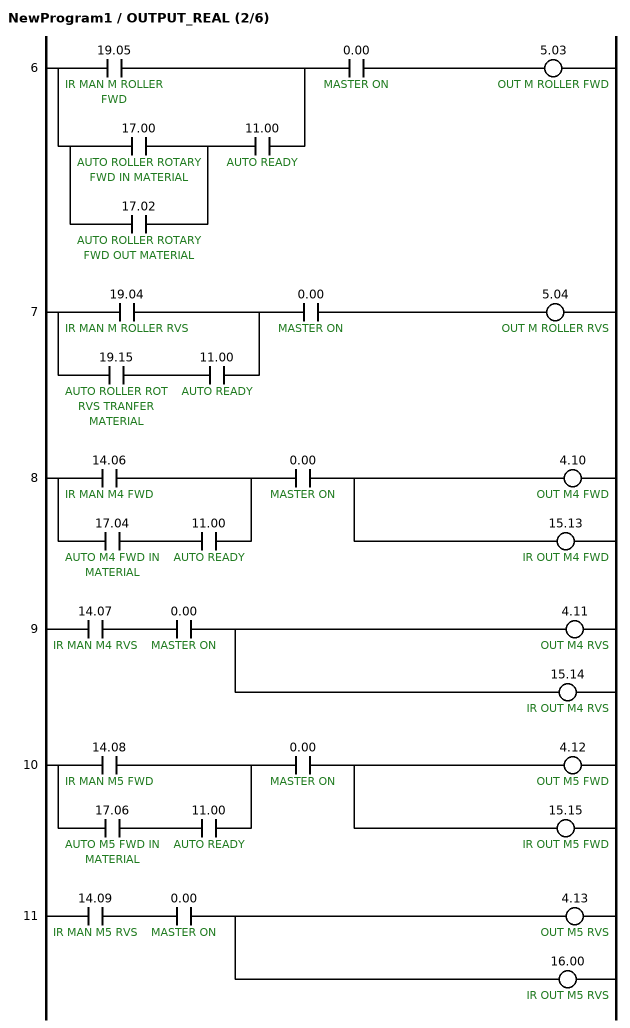
; [picture p24: NewProgram1 / OUTPUT_REAL, rungs 6-11]
; rung 6
LD 19.05  ; IR MAN M ROLLER FWD
LD 17.00  ; AUTO ROLLER ROTARY FWD IN MATERIAL
OR 17.02  ; AUTO ROLLER ROTARY FWD OUT MATERIAL
AND 11.00  ; AUTO READY
ORLD
AND 0.00  ; MASTER ON
OUT 5.03  ; OUT M ROLLER FWD
; rung 7
LD 19.04  ; IR MAN M ROLLER RVS
LD 19.15  ; AUTO ROLLER ROT RVS TRANFER MATERIAL
AND 11.00  ; AUTO READY
ORLD
AND 0.00  ; MASTER ON
OUT 5.04  ; OUT M ROLLER RVS
; rung 8
LD 14.06  ; IR MAN M4 FWD
LD 17.04  ; AUTO M4 FWD IN MATERIAL
AND 11.00  ; AUTO READY
ORLD
AND 0.00  ; MASTER ON
OUT 4.10  ; OUT M4 FWD
OUT 15.13  ; IR OUT M4 FWD
; rung 9
LD 14.07  ; IR MAN M4 RVS
AND 0.00  ; MASTER ON
OUT 4.11  ; OUT M4 RVS
OUT 15.14  ; IR OUT M4 RVS
; rung 10
LD 14.08  ; IR MAN M5 FWD
LD 17.06  ; AUTO M5 FWD IN MATERIAL
AND 11.00  ; AUTO READY
ORLD
AND 0.00  ; MASTER ON
OUT 4.12  ; OUT M5 FWD
OUT 15.15  ; IR OUT M5 FWD
; rung 11
LD 14.09  ; IR MAN M5 RVS
AND 0.00  ; MASTER ON
OUT 4.13  ; OUT M5 RVS
OUT 16.00  ; IR OUT M5 RVS

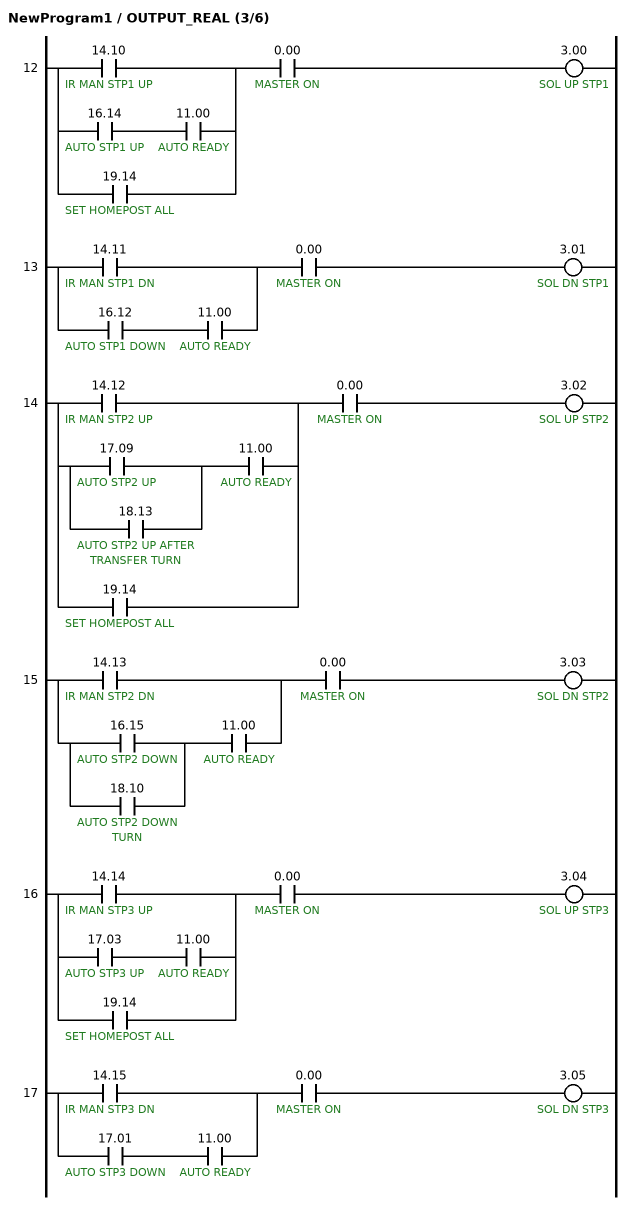
; rung 12
LD 14.10  ; IR MAN STP1 UP
LD 16.14  ; AUTO STP1 UP
AND 11.00  ; AUTO READY
ORLD
OR 19.14  ; SET HOMEPOST ALL
AND 0.00  ; MASTER ON
OUT 3.00  ; SOL UP STP1
; rung 13
LD 14.11  ; IR MAN STP1 DN
LD 16.12  ; AUTO STP1 DOWN
AND 11.00  ; AUTO READY
ORLD
AND 0.00  ; MASTER ON
OUT 3.01  ; SOL DN STP1
; rung 14
LD 14.12  ; IR MAN STP2 UP
LD 17.09  ; AUTO STP2 UP
OR 18.13  ; AUTO STP2 UP AFTER TRANSFER TURN
AND 11.00  ; AUTO READY
ORLD
OR 19.14  ; SET HOMEPOST ALL
AND 0.00  ; MASTER ON
OUT 3.02  ; SOL UP STP2
; rung 15
LD 14.13  ; IR MAN STP2 DN
LD 16.15  ; AUTO STP2 DOWN
OR 18.10  ; AUTO STP2 DOWN TURN
AND 11.00  ; AUTO READY
ORLD
AND 0.00  ; MASTER ON
OUT 3.03  ; SOL DN STP2
; rung 16
LD 14.14  ; IR MAN STP3 UP
LD 17.03  ; AUTO STP3 UP
AND 11.00  ; AUTO READY
ORLD
OR 19.14  ; SET HOMEPOST ALL
AND 0.00  ; MASTER ON
OUT 3.04  ; SOL UP STP3
; rung 17
LD 14.15  ; IR MAN STP3 DN
LD 17.01  ; AUTO STP3 DOWN
AND 11.00  ; AUTO READY
ORLD
AND 0.00  ; MASTER ON
OUT 3.05  ; SOL DN STP3

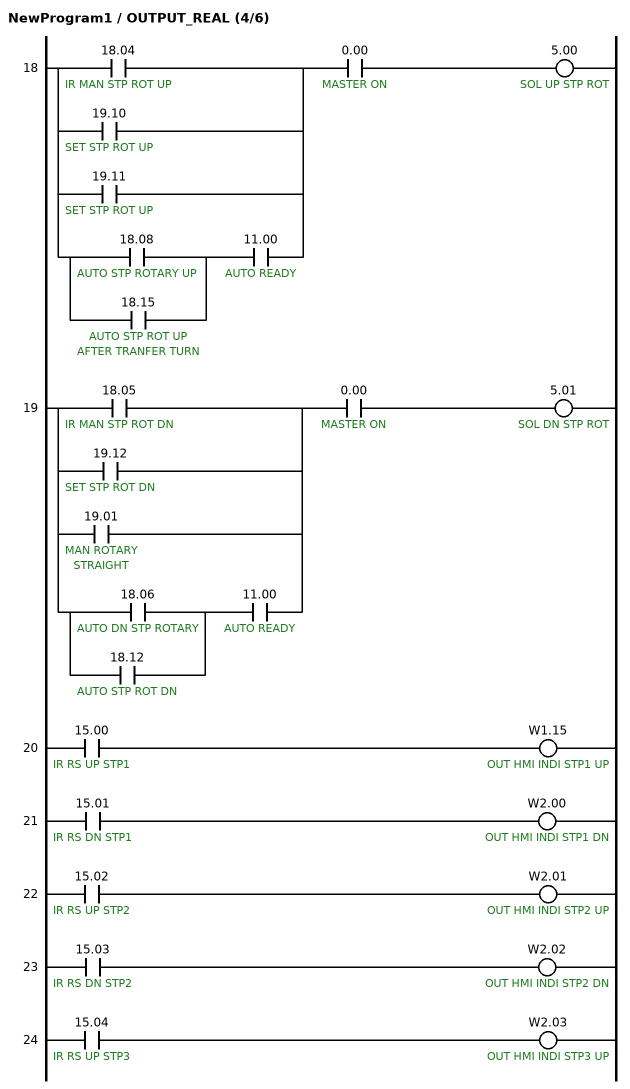
; rung 18
LD 18.04  ; IR MAN STP ROT UP
OR 19.10  ; SET STP ROT UP
OR 19.11  ; SET STP ROT UP
LD 18.08  ; AUTO STP ROTARY UP
OR 18.15  ; AUTO STP ROT UP AFTER TRANFER TURN
AND 11.00  ; AUTO READY
ORLD
AND 0.00  ; MASTER ON
OUT 5.00  ; SOL UP STP ROT
; rung 19
LD 18.05  ; IR MAN STP ROT DN
OR 19.12  ; SET STP ROT DN
OR 19.01  ; MAN ROTARY STRAIGHT
LD 18.06  ; AUTO DN STP ROTARY
OR 18.12  ; AUTO STP ROT DN
AND 11.00  ; AUTO READY
ORLD
AND 0.00  ; MASTER ON
OUT 5.01  ; SOL DN STP ROT
; rung 20
LD 15.00  ; IR RS UP STP1
OUT W1.15  ; OUT HMI INDI STP1 UP
; rung 21
LD 15.01  ; IR RS DN STP1
OUT W2.00  ; OUT HMI INDI STP1 DN
; rung 22
LD 15.02  ; IR RS UP STP2
OUT W2.01  ; OUT HMI INDI STP2 UP
; rung 23
LD 15.03  ; IR RS DN STP2
OUT W2.02  ; OUT HMI INDI STP2 DN
; rung 24
LD 15.04  ; IR RS UP STP3
OUT W2.03  ; OUT HMI INDI STP3 UP

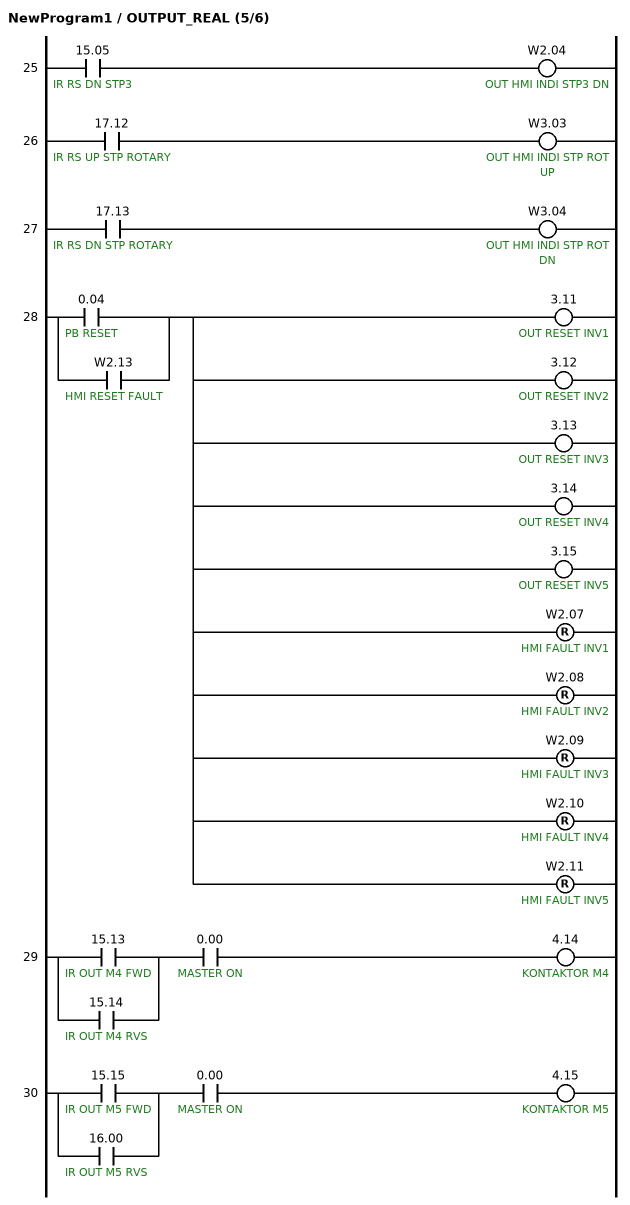
; rung 25
LD 15.05  ; IR RS DN STP3
OUT W2.04  ; OUT HMI INDI STP3 DN
; rung 26
LD 17.12  ; IR RS UP STP ROTARY
OUT W3.03  ; OUT HMI INDI STP ROT UP
; rung 27
LD 17.13  ; IR RS DN STP ROTARY
OUT W3.04  ; OUT HMI INDI STP ROT DN
; rung 28
LD 0.04  ; PB RESET
OR W2.13  ; HMI RESET FAULT
OUT 3.11  ; OUT RESET INV1
OUT 3.12  ; OUT RESET INV2
OUT 3.13  ; OUT RESET INV3
OUT 3.14  ; OUT RESET INV4
OUT 3.15  ; OUT RESET INV5
RSET W2.07  ; HMI FAULT INV1
RSET W2.08  ; HMI FAULT INV2
RSET W2.09  ; HMI FAULT INV3
RSET W2.10  ; HMI FAULT INV4
RSET W2.11  ; HMI FAULT INV5
; rung 29
LD 15.13  ; IR OUT M4 FWD
OR 15.14  ; IR OUT M4 RVS
AND 0.00  ; MASTER ON
OUT 4.14  ; KONTAKTOR M4
; rung 30
LD 15.15  ; IR OUT M5 FWD
OR 16.00  ; IR OUT M5 RVS
AND 0.00  ; MASTER ON
OUT 4.15  ; KONTAKTOR M5

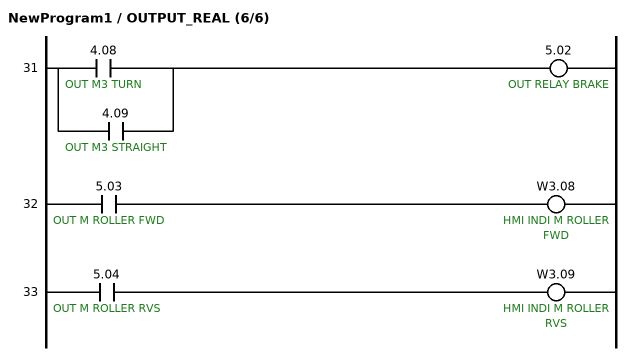
; rung 31
LD 4.08  ; OUT M3 TURN
OR 4.09  ; OUT M3 STRAIGHT
OUT 5.02  ; OUT RELAY BRAKE
; rung 32
LD 5.03  ; OUT M ROLLER FWD
OUT W3.08  ; HMI INDI M ROLLER FWD
; rung 33
LD 5.04  ; OUT M ROLLER RVS
OUT W3.09  ; HMI INDI M ROLLER RVS

### Section INPUT_REAL

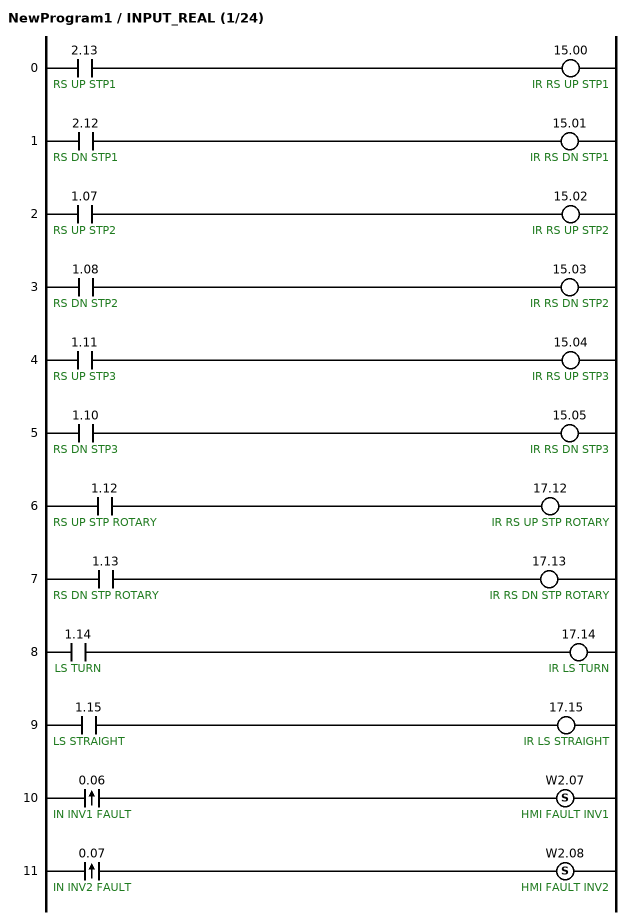
; rung 0
LD 2.13  ; RS UP STP1
OUT 15.00  ; IR RS UP STP1
; rung 1
LD 2.12  ; RS DN STP1
OUT 15.01  ; IR RS DN STP1
; rung 2
LD 1.07  ; RS UP STP2
OUT 15.02  ; IR RS UP STP2
; rung 3
LD 1.08  ; RS DN STP2
OUT 15.03  ; IR RS DN STP2
; rung 4
LD 1.11  ; RS UP STP3
OUT 15.04  ; IR RS UP STP3
; rung 5
LD 1.10  ; RS DN STP3
OUT 15.05  ; IR RS DN STP3
; rung 6
LD 1.12  ; RS UP STP ROTARY
OUT 17.12  ; IR RS UP STP ROTARY
; rung 7
LD 1.13  ; RS DN STP ROTARY
OUT 17.13  ; IR RS DN STP ROTARY
; rung 8
LD 1.14  ; LS TURN
OUT 17.14  ; IR LS TURN
; rung 9
LD 1.15  ; LS STRAIGHT
OUT 17.15  ; IR LS STRAIGHT
; rung 10
@LD 0.06  ; IN INV1 FAULT
SET W2.07  ; HMI FAULT INV1
; rung 11
@LD 0.07  ; IN INV2 FAULT
SET W2.08  ; HMI FAULT INV2

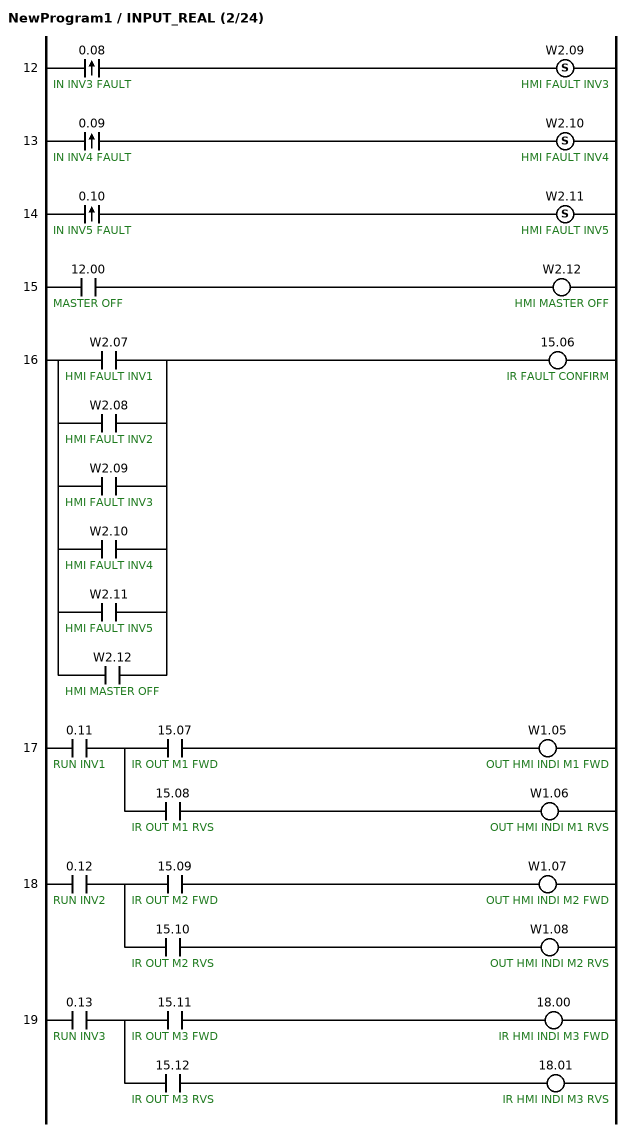
; rung 12
@LD 0.08  ; IN INV3 FAULT
SET W2.09  ; HMI FAULT INV3
; rung 13
@LD 0.09  ; IN INV4 FAULT
SET W2.10  ; HMI FAULT INV4
; rung 14
@LD 0.10  ; IN INV5 FAULT
SET W2.11  ; HMI FAULT INV5
; rung 15
LD 12.00  ; MASTER OFF
OUT W2.12  ; HMI MASTER OFF
; rung 16
LD W2.07  ; HMI FAULT INV1
OR W2.08  ; HMI FAULT INV2
OR W2.09  ; HMI FAULT INV3
OR W2.10  ; HMI FAULT INV4
OR W2.11  ; HMI FAULT INV5
OR W2.12  ; HMI MASTER OFF
OUT 15.06  ; IR FAULT CONFIRM
; rung 17
LD 0.11  ; RUN INV1
OUT TR0
AND 15.07  ; IR OUT M1 FWD
OUT W1.05  ; OUT HMI INDI M1 FWD
LD TR0
AND 15.08  ; IR OUT M1 RVS
OUT W1.06  ; OUT HMI INDI M1 RVS
; rung 18
LD 0.12  ; RUN INV2
OUT TR0
AND 15.09  ; IR OUT M2 FWD
OUT W1.07  ; OUT HMI INDI M2 FWD
LD TR0
AND 15.10  ; IR OUT M2 RVS
OUT W1.08  ; OUT HMI INDI M2 RVS
; rung 19
LD 0.13  ; RUN INV3
OUT TR0
AND 15.11  ; IR OUT M3 FWD
OUT 18.00  ; IR HMI INDI M3 FWD
LD TR0
AND 15.12  ; IR OUT M3 RVS
OUT 18.01  ; IR HMI INDI M3 RVS

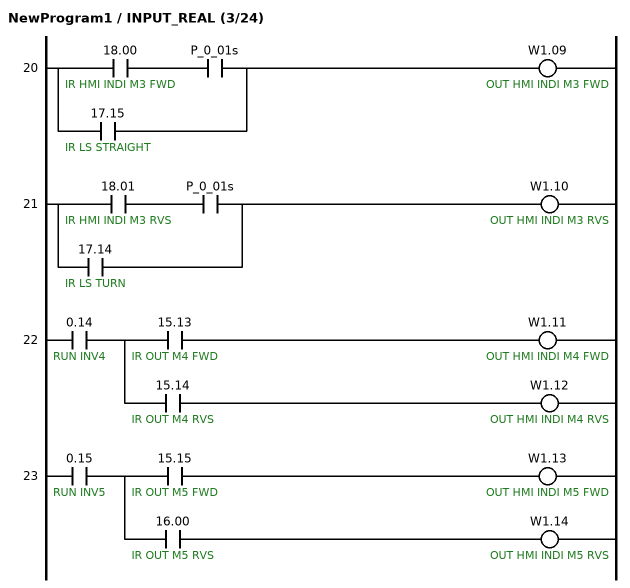
; rung 20
LD 18.00  ; IR HMI INDI M3 FWD
AND P_0_01s
OR 17.15  ; IR LS STRAIGHT
OUT W1.09  ; OUT HMI INDI M3 FWD
; rung 21
LD 18.01  ; IR HMI INDI M3 RVS
AND P_0_01s
OR 17.14  ; IR LS TURN
OUT W1.10  ; OUT HMI INDI M3 RVS
; rung 22
LD 0.14  ; RUN INV4
OUT TR0
AND 15.13  ; IR OUT M4 FWD
OUT W1.11  ; OUT HMI INDI M4 FWD
LD TR0
AND 15.14  ; IR OUT M4 RVS
OUT W1.12  ; OUT HMI INDI M4 RVS
; rung 23
LD 0.15  ; RUN INV5
OUT TR0
AND 15.15  ; IR OUT M5 FWD
OUT W1.13  ; OUT HMI INDI M5 FWD
LD TR0
AND 16.00  ; IR OUT M5 RVS
OUT W1.14  ; OUT HMI INDI M5 RVS

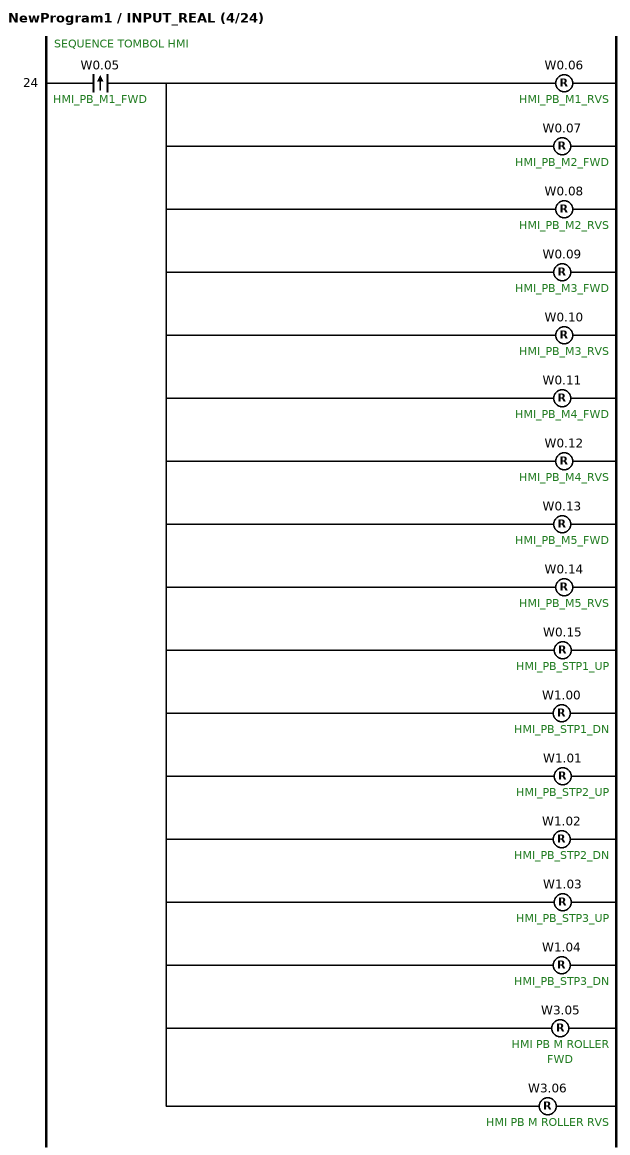
; rung 24: SEQUENCE TOMBOL HMI
@LD W0.05  ; HMI_PB_M1_FWD
RSET W0.06  ; HMI_PB_M1_RVS
RSET W0.07  ; HMI_PB_M2_FWD
RSET W0.08  ; HMI_PB_M2_RVS
RSET W0.09  ; HMI_PB_M3_FWD
RSET W0.10  ; HMI_PB_M3_RVS
RSET W0.11  ; HMI_PB_M4_FWD
RSET W0.12  ; HMI_PB_M4_RVS
RSET W0.13  ; HMI_PB_M5_FWD
RSET W0.14  ; HMI_PB_M5_RVS
RSET W0.15  ; HMI_PB_STP1_UP
RSET W1.00  ; HMI_PB_STP1_DN
RSET W1.01  ; HMI_PB_STP2_UP
RSET W1.02  ; HMI_PB_STP2_DN
RSET W1.03  ; HMI_PB_STP3_UP
RSET W1.04  ; HMI_PB_STP3_DN
RSET W3.05  ; HMI PB M ROLLER FWD
RSET W3.06  ; HMI PB M ROLLER RVS

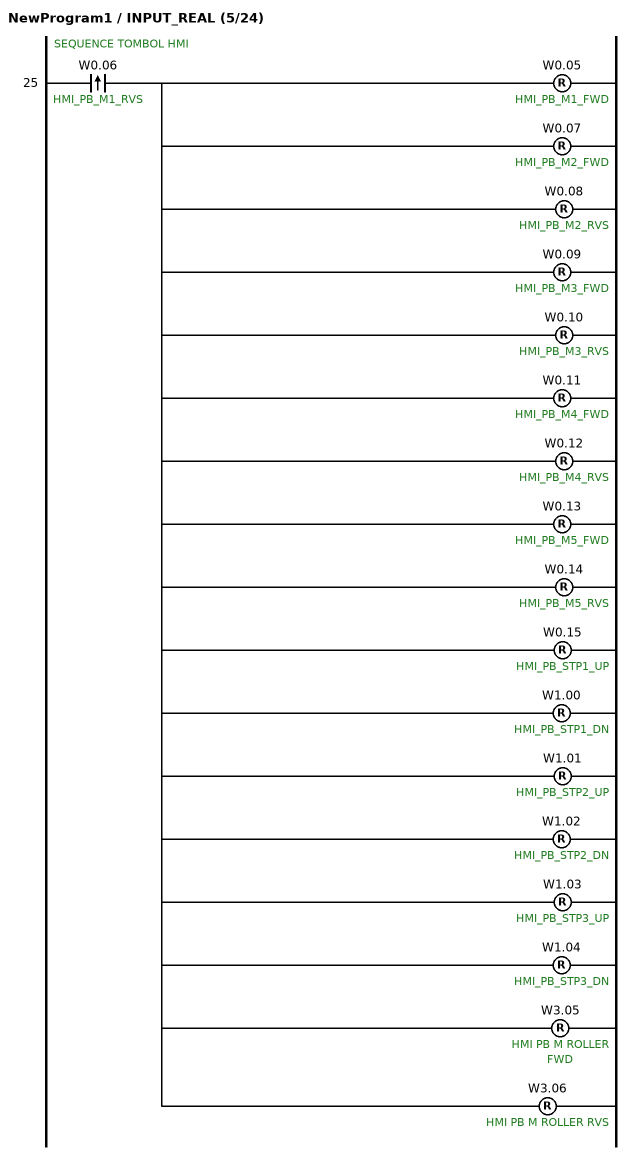
; rung 25: SEQUENCE TOMBOL HMI
@LD W0.06  ; HMI_PB_M1_RVS
RSET W0.05  ; HMI_PB_M1_FWD
RSET W0.07  ; HMI_PB_M2_FWD
RSET W0.08  ; HMI_PB_M2_RVS
RSET W0.09  ; HMI_PB_M3_FWD
RSET W0.10  ; HMI_PB_M3_RVS
RSET W0.11  ; HMI_PB_M4_FWD
RSET W0.12  ; HMI_PB_M4_RVS
RSET W0.13  ; HMI_PB_M5_FWD
RSET W0.14  ; HMI_PB_M5_RVS
RSET W0.15  ; HMI_PB_STP1_UP
RSET W1.00  ; HMI_PB_STP1_DN
RSET W1.01  ; HMI_PB_STP2_UP
RSET W1.02  ; HMI_PB_STP2_DN
RSET W1.03  ; HMI_PB_STP3_UP
RSET W1.04  ; HMI_PB_STP3_DN
RSET W3.05  ; HMI PB M ROLLER FWD
RSET W3.06  ; HMI PB M ROLLER RVS

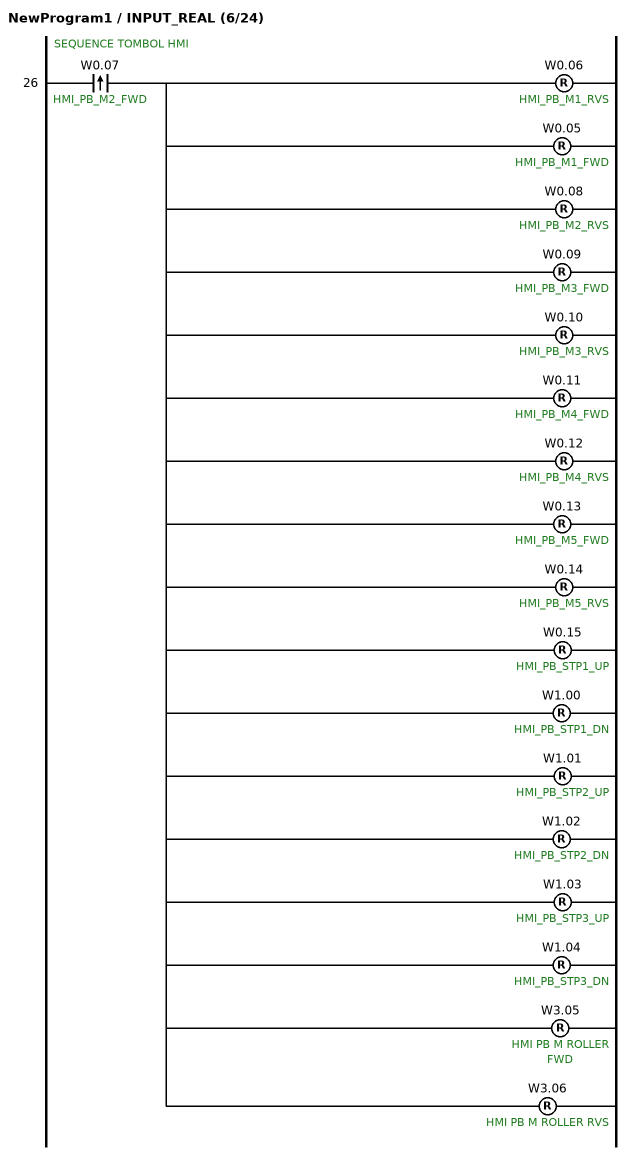
; rung 26: SEQUENCE TOMBOL HMI
@LD W0.07  ; HMI_PB_M2_FWD
RSET W0.06  ; HMI_PB_M1_RVS
RSET W0.05  ; HMI_PB_M1_FWD
RSET W0.08  ; HMI_PB_M2_RVS
RSET W0.09  ; HMI_PB_M3_FWD
RSET W0.10  ; HMI_PB_M3_RVS
RSET W0.11  ; HMI_PB_M4_FWD
RSET W0.12  ; HMI_PB_M4_RVS
RSET W0.13  ; HMI_PB_M5_FWD
RSET W0.14  ; HMI_PB_M5_RVS
RSET W0.15  ; HMI_PB_STP1_UP
RSET W1.00  ; HMI_PB_STP1_DN
RSET W1.01  ; HMI_PB_STP2_UP
RSET W1.02  ; HMI_PB_STP2_DN
RSET W1.03  ; HMI_PB_STP3_UP
RSET W1.04  ; HMI_PB_STP3_DN
RSET W3.05  ; HMI PB M ROLLER FWD
RSET W3.06  ; HMI PB M ROLLER RVS

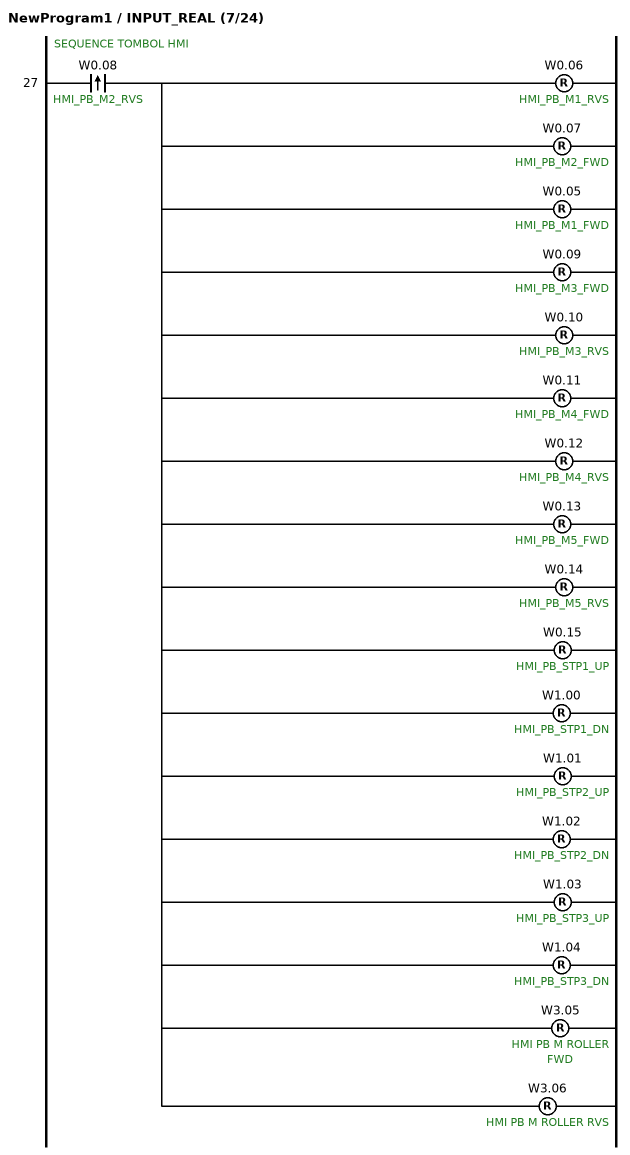
; rung 27: SEQUENCE TOMBOL HMI
@LD W0.08  ; HMI_PB_M2_RVS
RSET W0.06  ; HMI_PB_M1_RVS
RSET W0.07  ; HMI_PB_M2_FWD
RSET W0.05  ; HMI_PB_M1_FWD
RSET W0.09  ; HMI_PB_M3_FWD
RSET W0.10  ; HMI_PB_M3_RVS
RSET W0.11  ; HMI_PB_M4_FWD
RSET W0.12  ; HMI_PB_M4_RVS
RSET W0.13  ; HMI_PB_M5_FWD
RSET W0.14  ; HMI_PB_M5_RVS
RSET W0.15  ; HMI_PB_STP1_UP
RSET W1.00  ; HMI_PB_STP1_DN
RSET W1.01  ; HMI_PB_STP2_UP
RSET W1.02  ; HMI_PB_STP2_DN
RSET W1.03  ; HMI_PB_STP3_UP
RSET W1.04  ; HMI_PB_STP3_DN
RSET W3.05  ; HMI PB M ROLLER FWD
RSET W3.06  ; HMI PB M ROLLER RVS

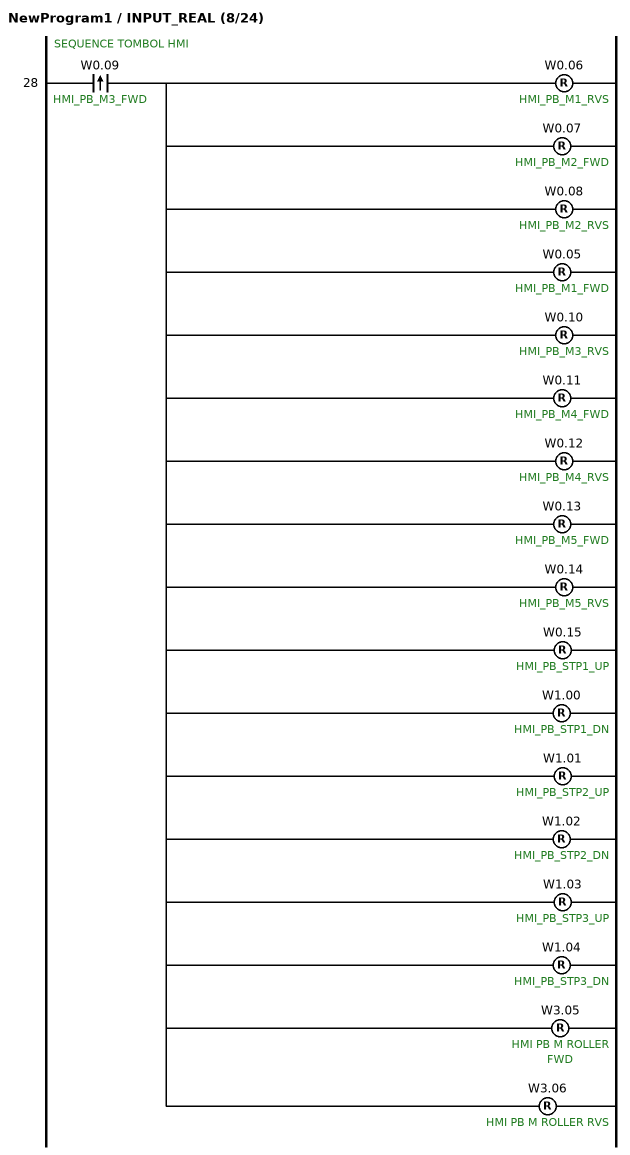
; rung 28: SEQUENCE TOMBOL HMI
@LD W0.09  ; HMI_PB_M3_FWD
RSET W0.06  ; HMI_PB_M1_RVS
RSET W0.07  ; HMI_PB_M2_FWD
RSET W0.08  ; HMI_PB_M2_RVS
RSET W0.05  ; HMI_PB_M1_FWD
RSET W0.10  ; HMI_PB_M3_RVS
RSET W0.11  ; HMI_PB_M4_FWD
RSET W0.12  ; HMI_PB_M4_RVS
RSET W0.13  ; HMI_PB_M5_FWD
RSET W0.14  ; HMI_PB_M5_RVS
RSET W0.15  ; HMI_PB_STP1_UP
RSET W1.00  ; HMI_PB_STP1_DN
RSET W1.01  ; HMI_PB_STP2_UP
RSET W1.02  ; HMI_PB_STP2_DN
RSET W1.03  ; HMI_PB_STP3_UP
RSET W1.04  ; HMI_PB_STP3_DN
RSET W3.05  ; HMI PB M ROLLER FWD
RSET W3.06  ; HMI PB M ROLLER RVS

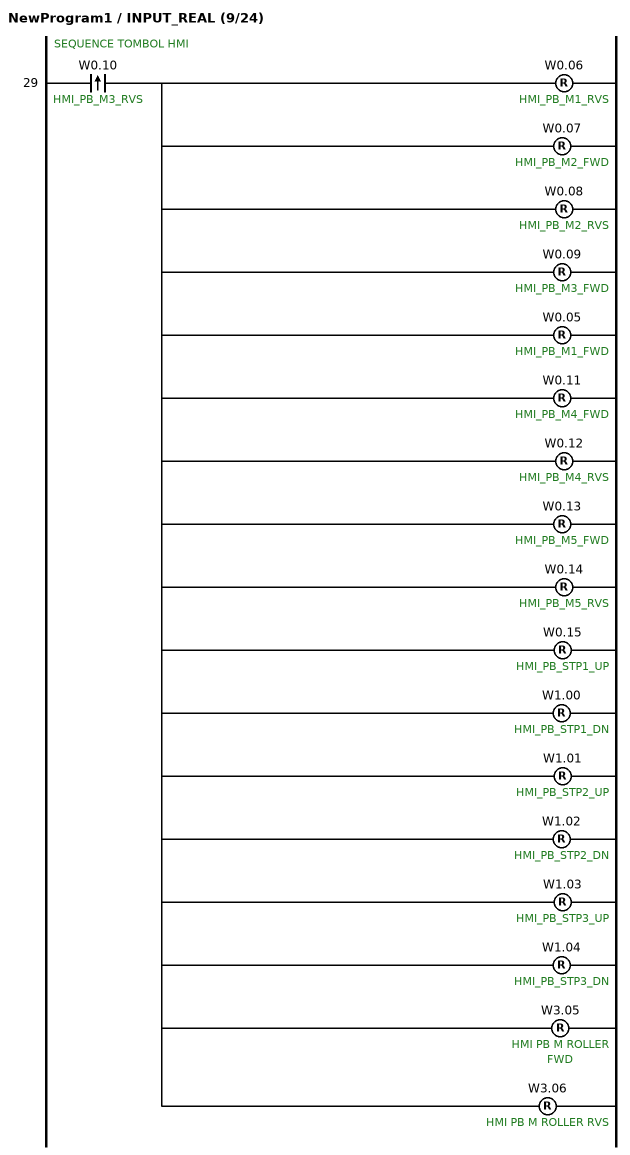
; rung 29: SEQUENCE TOMBOL HMI
@LD W0.10  ; HMI_PB_M3_RVS
RSET W0.06  ; HMI_PB_M1_RVS
RSET W0.07  ; HMI_PB_M2_FWD
RSET W0.08  ; HMI_PB_M2_RVS
RSET W0.09  ; HMI_PB_M3_FWD
RSET W0.05  ; HMI_PB_M1_FWD
RSET W0.11  ; HMI_PB_M4_FWD
RSET W0.12  ; HMI_PB_M4_RVS
RSET W0.13  ; HMI_PB_M5_FWD
RSET W0.14  ; HMI_PB_M5_RVS
RSET W0.15  ; HMI_PB_STP1_UP
RSET W1.00  ; HMI_PB_STP1_DN
RSET W1.01  ; HMI_PB_STP2_UP
RSET W1.02  ; HMI_PB_STP2_DN
RSET W1.03  ; HMI_PB_STP3_UP
RSET W1.04  ; HMI_PB_STP3_DN
RSET W3.05  ; HMI PB M ROLLER FWD
RSET W3.06  ; HMI PB M ROLLER RVS

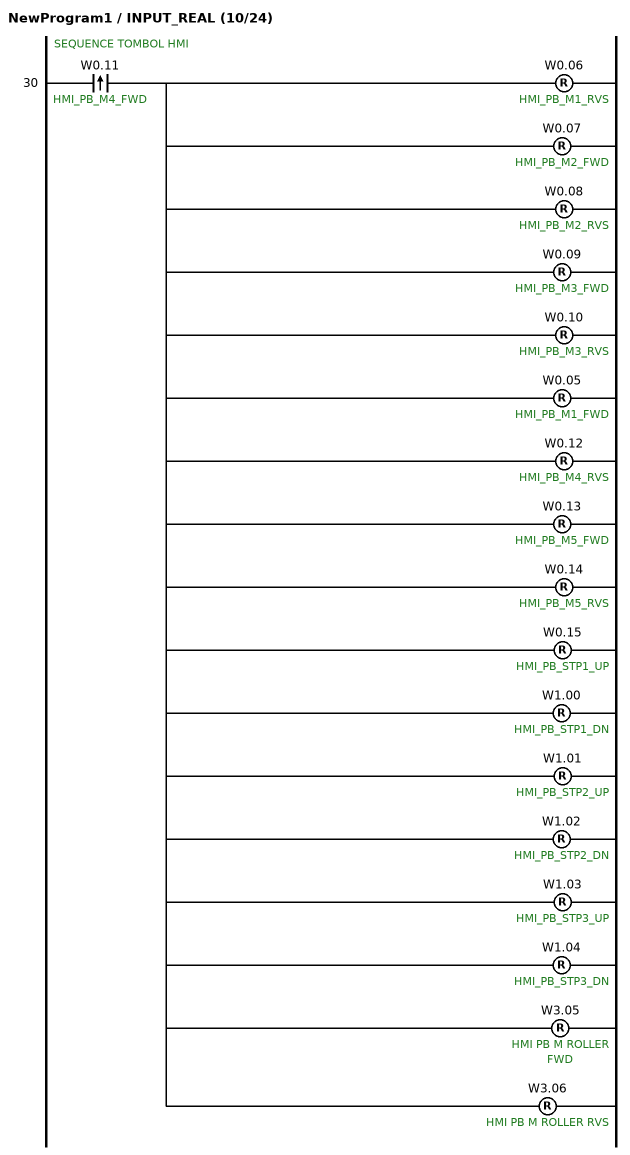
; rung 30: SEQUENCE TOMBOL HMI
@LD W0.11  ; HMI_PB_M4_FWD
RSET W0.06  ; HMI_PB_M1_RVS
RSET W0.07  ; HMI_PB_M2_FWD
RSET W0.08  ; HMI_PB_M2_RVS
RSET W0.09  ; HMI_PB_M3_FWD
RSET W0.10  ; HMI_PB_M3_RVS
RSET W0.05  ; HMI_PB_M1_FWD
RSET W0.12  ; HMI_PB_M4_RVS
RSET W0.13  ; HMI_PB_M5_FWD
RSET W0.14  ; HMI_PB_M5_RVS
RSET W0.15  ; HMI_PB_STP1_UP
RSET W1.00  ; HMI_PB_STP1_DN
RSET W1.01  ; HMI_PB_STP2_UP
RSET W1.02  ; HMI_PB_STP2_DN
RSET W1.03  ; HMI_PB_STP3_UP
RSET W1.04  ; HMI_PB_STP3_DN
RSET W3.05  ; HMI PB M ROLLER FWD
RSET W3.06  ; HMI PB M ROLLER RVS

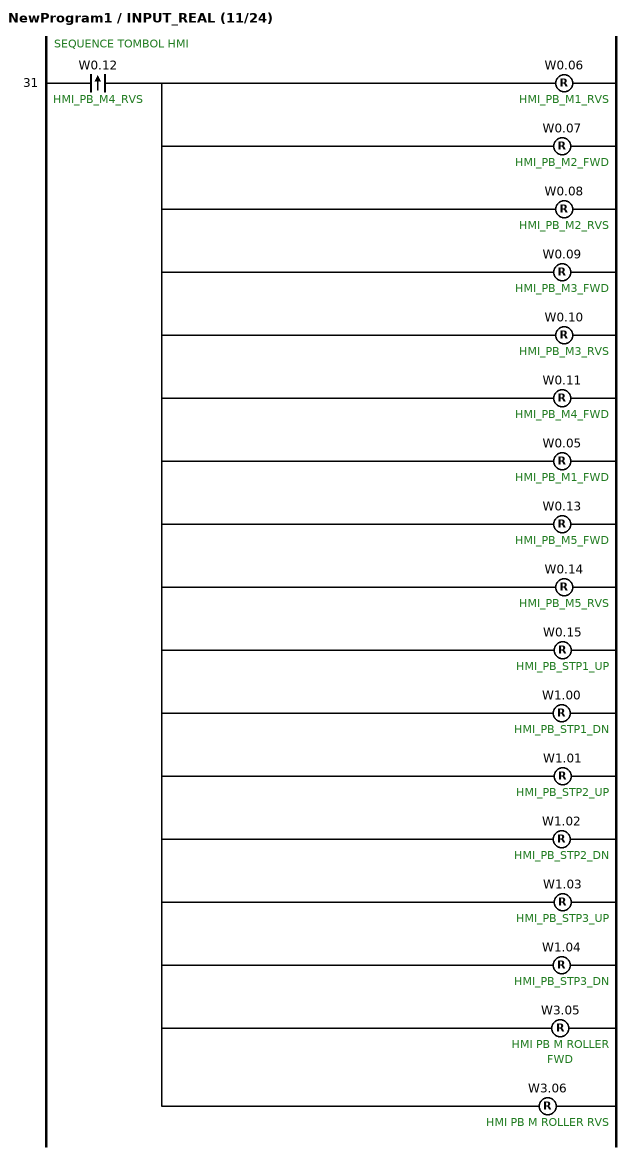
; rung 31: SEQUENCE TOMBOL HMI
@LD W0.12  ; HMI_PB_M4_RVS
RSET W0.06  ; HMI_PB_M1_RVS
RSET W0.07  ; HMI_PB_M2_FWD
RSET W0.08  ; HMI_PB_M2_RVS
RSET W0.09  ; HMI_PB_M3_FWD
RSET W0.10  ; HMI_PB_M3_RVS
RSET W0.11  ; HMI_PB_M4_FWD
RSET W0.05  ; HMI_PB_M1_FWD
RSET W0.13  ; HMI_PB_M5_FWD
RSET W0.14  ; HMI_PB_M5_RVS
RSET W0.15  ; HMI_PB_STP1_UP
RSET W1.00  ; HMI_PB_STP1_DN
RSET W1.01  ; HMI_PB_STP2_UP
RSET W1.02  ; HMI_PB_STP2_DN
RSET W1.03  ; HMI_PB_STP3_UP
RSET W1.04  ; HMI_PB_STP3_DN
RSET W3.05  ; HMI PB M ROLLER FWD
RSET W3.06  ; HMI PB M ROLLER RVS

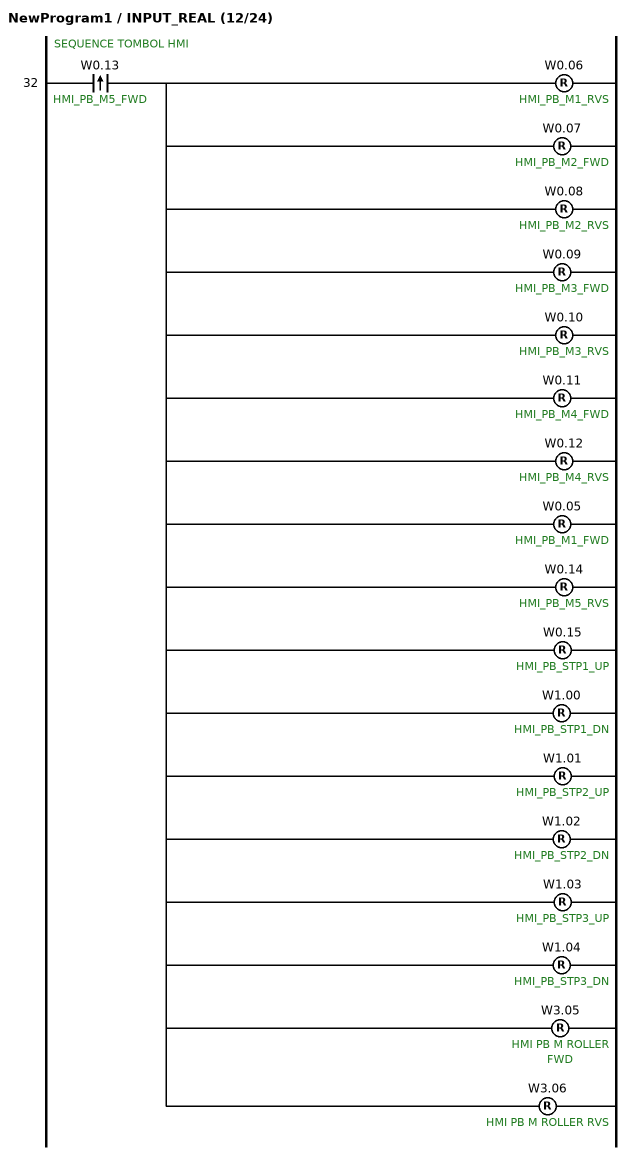
; rung 32: SEQUENCE TOMBOL HMI
@LD W0.13  ; HMI_PB_M5_FWD
RSET W0.06  ; HMI_PB_M1_RVS
RSET W0.07  ; HMI_PB_M2_FWD
RSET W0.08  ; HMI_PB_M2_RVS
RSET W0.09  ; HMI_PB_M3_FWD
RSET W0.10  ; HMI_PB_M3_RVS
RSET W0.11  ; HMI_PB_M4_FWD
RSET W0.12  ; HMI_PB_M4_RVS
RSET W0.05  ; HMI_PB_M1_FWD
RSET W0.14  ; HMI_PB_M5_RVS
RSET W0.15  ; HMI_PB_STP1_UP
RSET W1.00  ; HMI_PB_STP1_DN
RSET W1.01  ; HMI_PB_STP2_UP
RSET W1.02  ; HMI_PB_STP2_DN
RSET W1.03  ; HMI_PB_STP3_UP
RSET W1.04  ; HMI_PB_STP3_DN
RSET W3.05  ; HMI PB M ROLLER FWD
RSET W3.06  ; HMI PB M ROLLER RVS

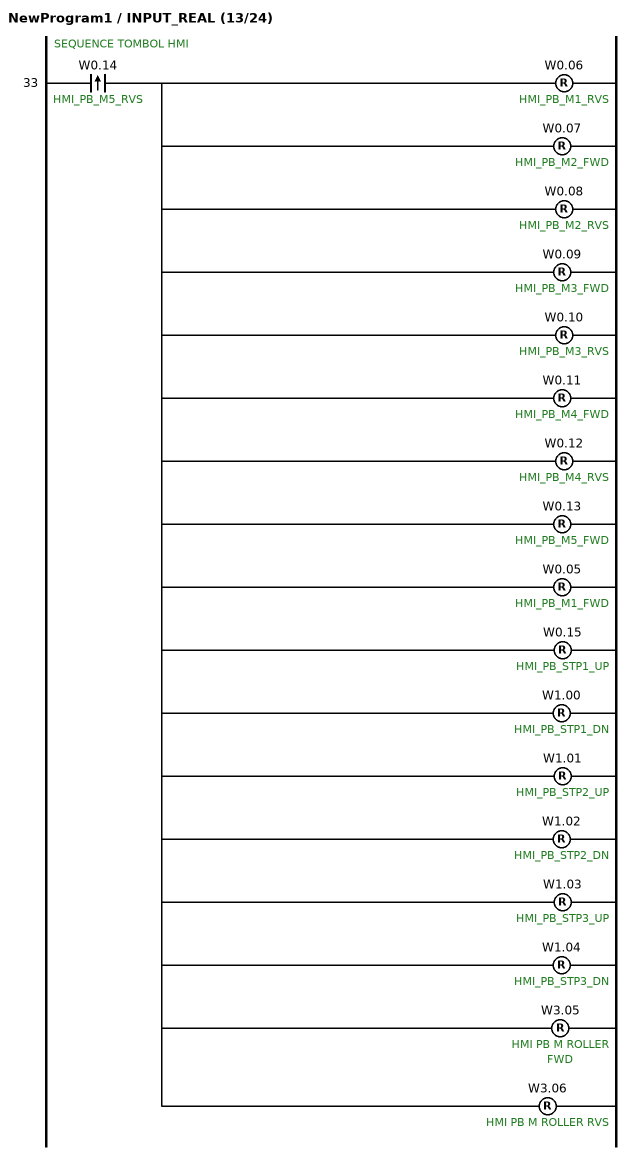
; rung 33: SEQUENCE TOMBOL HMI
@LD W0.14  ; HMI_PB_M5_RVS
RSET W0.06  ; HMI_PB_M1_RVS
RSET W0.07  ; HMI_PB_M2_FWD
RSET W0.08  ; HMI_PB_M2_RVS
RSET W0.09  ; HMI_PB_M3_FWD
RSET W0.10  ; HMI_PB_M3_RVS
RSET W0.11  ; HMI_PB_M4_FWD
RSET W0.12  ; HMI_PB_M4_RVS
RSET W0.13  ; HMI_PB_M5_FWD
RSET W0.05  ; HMI_PB_M1_FWD
RSET W0.15  ; HMI_PB_STP1_UP
RSET W1.00  ; HMI_PB_STP1_DN
RSET W1.01  ; HMI_PB_STP2_UP
RSET W1.02  ; HMI_PB_STP2_DN
RSET W1.03  ; HMI_PB_STP3_UP
RSET W1.04  ; HMI_PB_STP3_DN
RSET W3.05  ; HMI PB M ROLLER FWD
RSET W3.06  ; HMI PB M ROLLER RVS

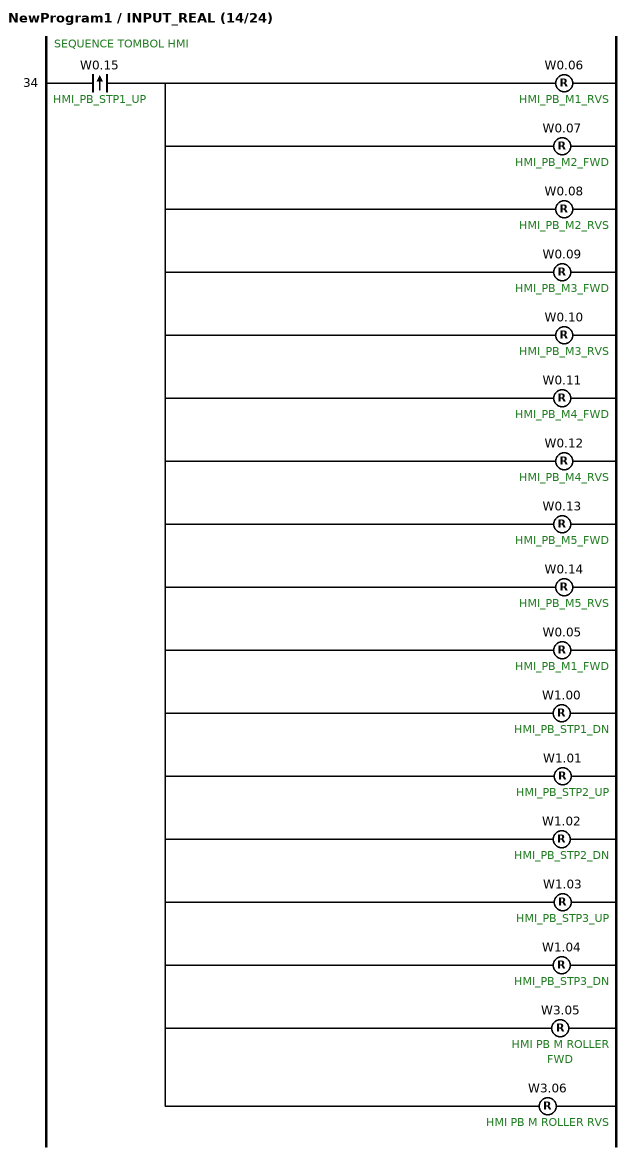
; rung 34: SEQUENCE TOMBOL HMI
@LD W0.15  ; HMI_PB_STP1_UP
RSET W0.06  ; HMI_PB_M1_RVS
RSET W0.07  ; HMI_PB_M2_FWD
RSET W0.08  ; HMI_PB_M2_RVS
RSET W0.09  ; HMI_PB_M3_FWD
RSET W0.10  ; HMI_PB_M3_RVS
RSET W0.11  ; HMI_PB_M4_FWD
RSET W0.12  ; HMI_PB_M4_RVS
RSET W0.13  ; HMI_PB_M5_FWD
RSET W0.14  ; HMI_PB_M5_RVS
RSET W0.05  ; HMI_PB_M1_FWD
RSET W1.00  ; HMI_PB_STP1_DN
RSET W1.01  ; HMI_PB_STP2_UP
RSET W1.02  ; HMI_PB_STP2_DN
RSET W1.03  ; HMI_PB_STP3_UP
RSET W1.04  ; HMI_PB_STP3_DN
RSET W3.05  ; HMI PB M ROLLER FWD
RSET W3.06  ; HMI PB M ROLLER RVS

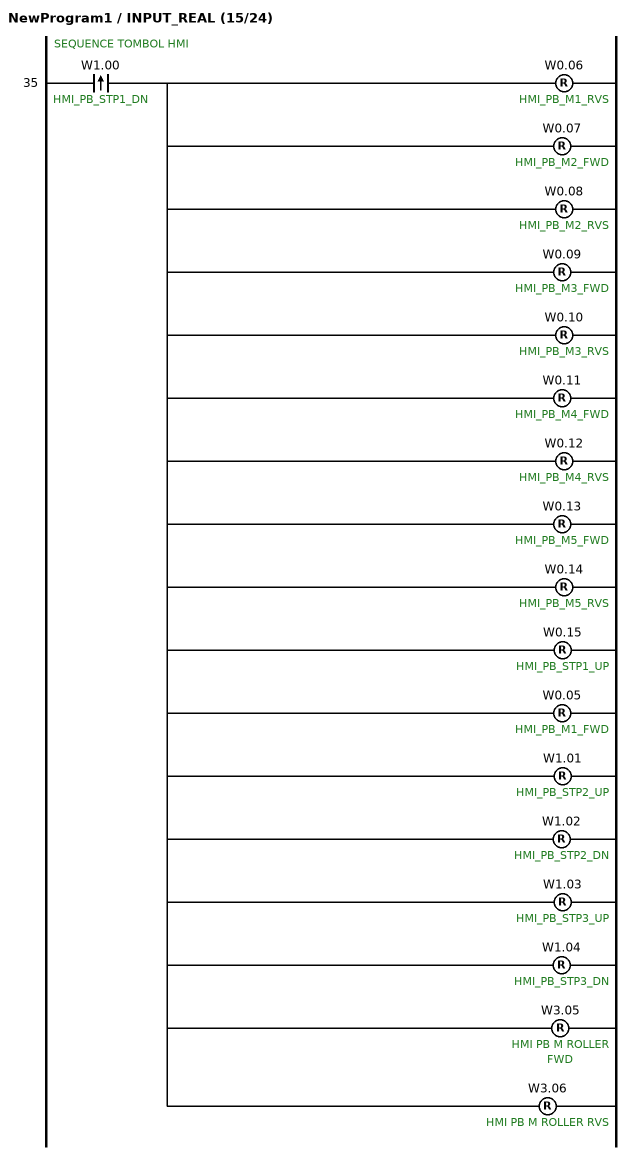
; rung 35: SEQUENCE TOMBOL HMI
@LD W1.00  ; HMI_PB_STP1_DN
RSET W0.06  ; HMI_PB_M1_RVS
RSET W0.07  ; HMI_PB_M2_FWD
RSET W0.08  ; HMI_PB_M2_RVS
RSET W0.09  ; HMI_PB_M3_FWD
RSET W0.10  ; HMI_PB_M3_RVS
RSET W0.11  ; HMI_PB_M4_FWD
RSET W0.12  ; HMI_PB_M4_RVS
RSET W0.13  ; HMI_PB_M5_FWD
RSET W0.14  ; HMI_PB_M5_RVS
RSET W0.15  ; HMI_PB_STP1_UP
RSET W0.05  ; HMI_PB_M1_FWD
RSET W1.01  ; HMI_PB_STP2_UP
RSET W1.02  ; HMI_PB_STP2_DN
RSET W1.03  ; HMI_PB_STP3_UP
RSET W1.04  ; HMI_PB_STP3_DN
RSET W3.05  ; HMI PB M ROLLER FWD
RSET W3.06  ; HMI PB M ROLLER RVS

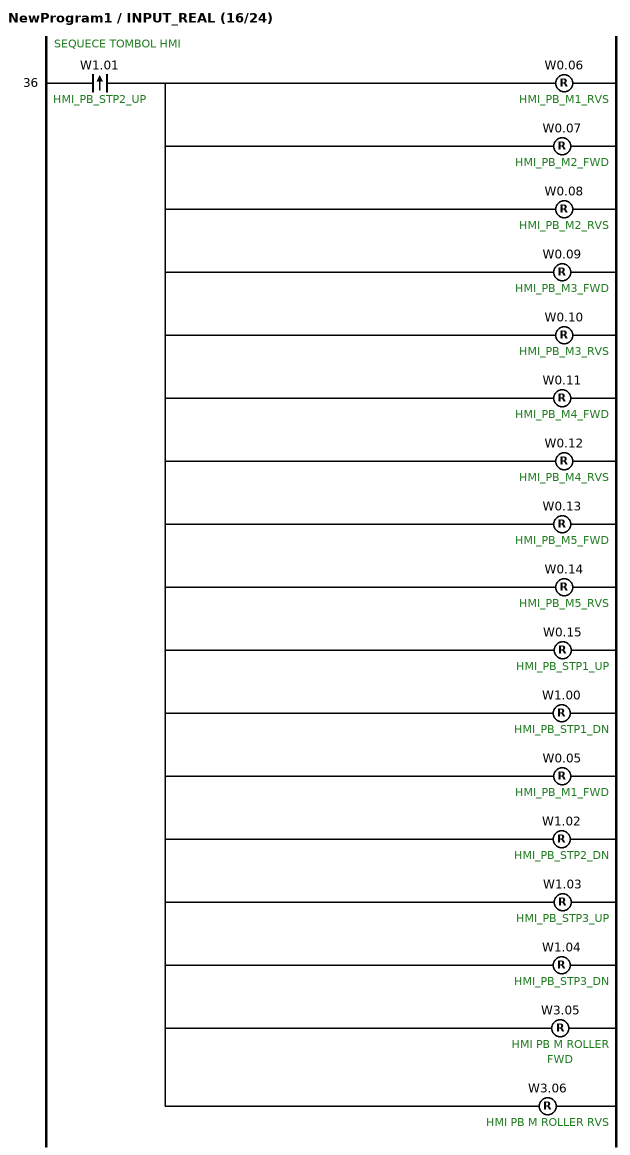
; rung 36: SEQUECE TOMBOL HMI
@LD W1.01  ; HMI_PB_STP2_UP
RSET W0.06  ; HMI_PB_M1_RVS
RSET W0.07  ; HMI_PB_M2_FWD
RSET W0.08  ; HMI_PB_M2_RVS
RSET W0.09  ; HMI_PB_M3_FWD
RSET W0.10  ; HMI_PB_M3_RVS
RSET W0.11  ; HMI_PB_M4_FWD
RSET W0.12  ; HMI_PB_M4_RVS
RSET W0.13  ; HMI_PB_M5_FWD
RSET W0.14  ; HMI_PB_M5_RVS
RSET W0.15  ; HMI_PB_STP1_UP
RSET W1.00  ; HMI_PB_STP1_DN
RSET W0.05  ; HMI_PB_M1_FWD
RSET W1.02  ; HMI_PB_STP2_DN
RSET W1.03  ; HMI_PB_STP3_UP
RSET W1.04  ; HMI_PB_STP3_DN
RSET W3.05  ; HMI PB M ROLLER FWD
RSET W3.06  ; HMI PB M ROLLER RVS

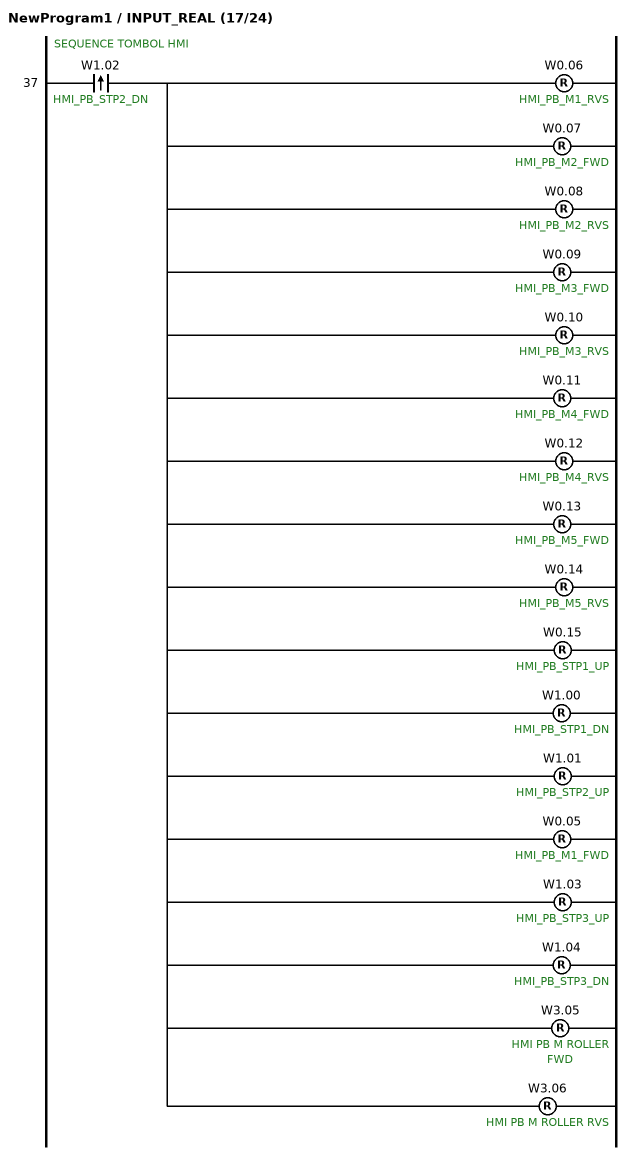
; rung 37: SEQUENCE TOMBOL HMI
@LD W1.02  ; HMI_PB_STP2_DN
RSET W0.06  ; HMI_PB_M1_RVS
RSET W0.07  ; HMI_PB_M2_FWD
RSET W0.08  ; HMI_PB_M2_RVS
RSET W0.09  ; HMI_PB_M3_FWD
RSET W0.10  ; HMI_PB_M3_RVS
RSET W0.11  ; HMI_PB_M4_FWD
RSET W0.12  ; HMI_PB_M4_RVS
RSET W0.13  ; HMI_PB_M5_FWD
RSET W0.14  ; HMI_PB_M5_RVS
RSET W0.15  ; HMI_PB_STP1_UP
RSET W1.00  ; HMI_PB_STP1_DN
RSET W1.01  ; HMI_PB_STP2_UP
RSET W0.05  ; HMI_PB_M1_FWD
RSET W1.03  ; HMI_PB_STP3_UP
RSET W1.04  ; HMI_PB_STP3_DN
RSET W3.05  ; HMI PB M ROLLER FWD
RSET W3.06  ; HMI PB M ROLLER RVS

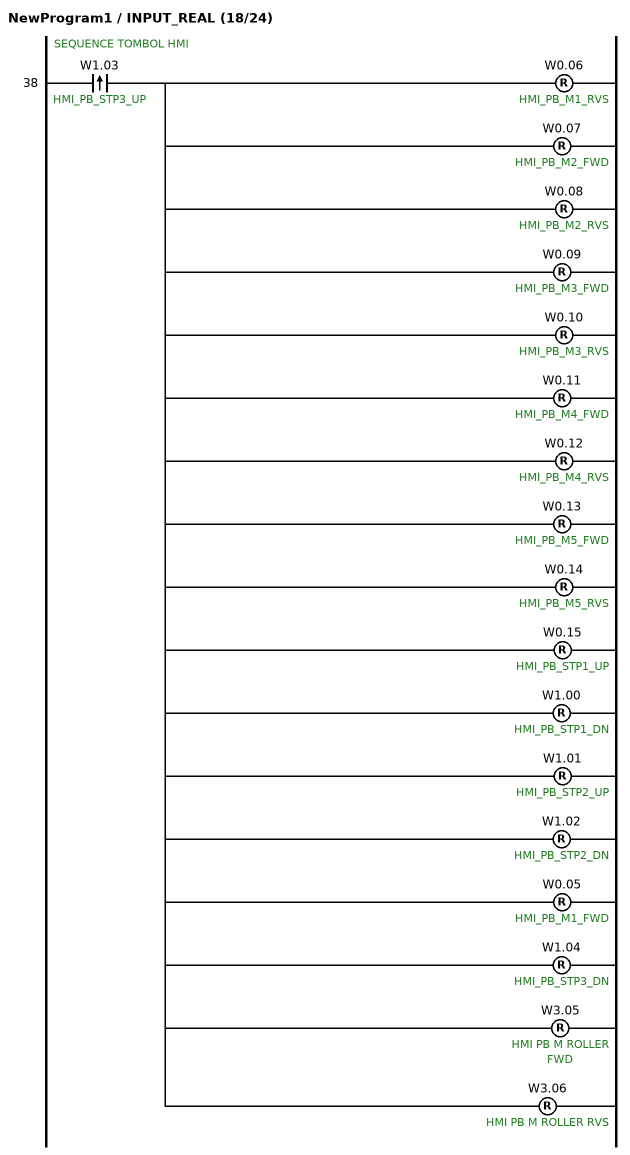
; rung 38: SEQUENCE TOMBOL HMI
@LD W1.03  ; HMI_PB_STP3_UP
RSET W0.06  ; HMI_PB_M1_RVS
RSET W0.07  ; HMI_PB_M2_FWD
RSET W0.08  ; HMI_PB_M2_RVS
RSET W0.09  ; HMI_PB_M3_FWD
RSET W0.10  ; HMI_PB_M3_RVS
RSET W0.11  ; HMI_PB_M4_FWD
RSET W0.12  ; HMI_PB_M4_RVS
RSET W0.13  ; HMI_PB_M5_FWD
RSET W0.14  ; HMI_PB_M5_RVS
RSET W0.15  ; HMI_PB_STP1_UP
RSET W1.00  ; HMI_PB_STP1_DN
RSET W1.01  ; HMI_PB_STP2_UP
RSET W1.02  ; HMI_PB_STP2_DN
RSET W0.05  ; HMI_PB_M1_FWD
RSET W1.04  ; HMI_PB_STP3_DN
RSET W3.05  ; HMI PB M ROLLER FWD
RSET W3.06  ; HMI PB M ROLLER RVS

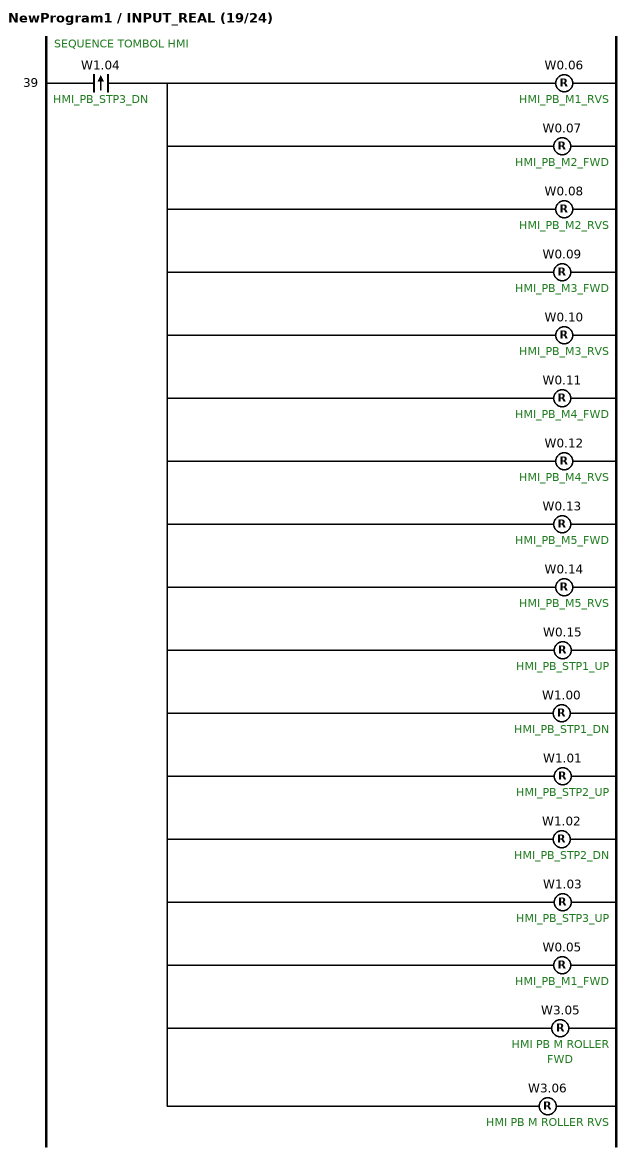
; rung 39: SEQUENCE TOMBOL HMI
@LD W1.04  ; HMI_PB_STP3_DN
RSET W0.06  ; HMI_PB_M1_RVS
RSET W0.07  ; HMI_PB_M2_FWD
RSET W0.08  ; HMI_PB_M2_RVS
RSET W0.09  ; HMI_PB_M3_FWD
RSET W0.10  ; HMI_PB_M3_RVS
RSET W0.11  ; HMI_PB_M4_FWD
RSET W0.12  ; HMI_PB_M4_RVS
RSET W0.13  ; HMI_PB_M5_FWD
RSET W0.14  ; HMI_PB_M5_RVS
RSET W0.15  ; HMI_PB_STP1_UP
RSET W1.00  ; HMI_PB_STP1_DN
RSET W1.01  ; HMI_PB_STP2_UP
RSET W1.02  ; HMI_PB_STP2_DN
RSET W1.03  ; HMI_PB_STP3_UP
RSET W0.05  ; HMI_PB_M1_FWD
RSET W3.05  ; HMI PB M ROLLER FWD
RSET W3.06  ; HMI PB M ROLLER RVS

